Fanuc KAREL source: KT00500.KL

PROGRAM KT00500
%NOLOCKGROUP
VAR
  P1: XYZWPR
  P2: XYZWPR
  OUT: XYZWPR
BEGIN
  P1.X = 1.0
  P2.Y = 2.0
  P1.X = 1.0
  P2.Y = 2.0
  OUT = P1 : P2
END KT00500
